// Mitsubishi GX Works2 project: PLC_GROUP2   PLC: FX3G

// global labels: Global1
VAR_GLOBAL
  start_day AT X007 : BOOL;
  Input_Oats AT D1100 : REAL;
  Oats AT D1101 : REAL;
  Input_Pro AT D2100 : REAL;
  Pro AT D2101 : REAL;
  Input_Honey AT D3100 : REAL;
  Honey AT D3101 : REAL;
  work_on AT Y000 : BOOL;
  work_off AT M0 : BOOL;
  end_pack AT M10 : BOOL;
END_VAR
VAR_GLOBAL CONSTANT
  classic_min_pro : REAL := 160;
  classic_min_honey : REAL := 120;
END_VAR
VAR_GLOBAL
  start_mix AT X003 : BOOL;
  Classic AT M16 : BOOL;
  Protein AT M18 : BOOL;
  cannot_mix AT M1 : BOOL;
END_VAR
VAR_GLOBAL CONSTANT
  normalizer : INT := 400;
  max_classic : REAL := 5;
END_VAR
VAR_GLOBAL
  timer_mix_5 AT TC1 : BOOL;
  timer_mix_finish AT TS1 : BOOL;
  mixing AT Y003 : BOOL;
END_VAR
VAR_GLOBAL CONSTANT
  sub_400 : REAL := 400.0;
  sub_160 : REAL := 160.0;
  sub_120 : REAL := 120.0;
  sub_240 : REAL := 240.0;
  sub_320 : REAL := 320.0;
END_VAR
VAR_GLOBAL
  mix_finish AT M8 : BOOL;
  start_bake AT X002 : BOOL;
  finish_bake AT M12 : BOOL;
  timer_bake_classic AT TC2 : BOOL;
END_VAR
VAR_GLOBAL CONSTANT
  four_sec : INT := 40;
END_VAR
VAR_GLOBAL
  timer_bake_pro AT TC3 : BOOL;
END_VAR
VAR_GLOBAL CONSTANT
  five_sec : INT := 50;
END_VAR
VAR_GLOBAL
  timer_bake_classic_finish AT TS2 : BOOL;
  timer_bake_pro_finish AT TS3 : BOOL;
  bake_in_process AT M20 : BOOL;
  timer_bake1 AT TC4 : BOOL;
END_VAR
VAR_GLOBAL CONSTANT
  flashing : INT := 005;
END_VAR
VAR_GLOBAL
  timer_bake1_finish AT TS4 : BOOL;
  lamp1 AT Y001 : BOOL;
  timer_bake2 AT TC5 : BOOL;
  lamp2 AT Y002 : BOOL;
  timer_bake2_finish AT TS5 : BOOL;
  start_pack AT X006 : BOOL;
  pack_hatif AT X000 : BOOL;
  counter_pack AT CC1 : BOOL;
END_VAR
VAR_GLOBAL CONSTANT
  eight_hatifim : INT := 8;
END_VAR
VAR_GLOBAL
  hatifim_packed AT CN1 : INT;
END_VAR
VAR_GLOBAL CONSTANT
  zero : INT;
END_VAR
VAR_GLOBAL
  new_pack AT M30 : BOOL;
  lamp4 AT Y004 : BOOL;
  counter_pack_finish AT CS1 : BOOL;
END_VAR
VAR_GLOBAL CONSTANT
  add_one_pack : INT := 1;
END_VAR
VAR_GLOBAL
  emergency AT X005 : BOOL;
END_VAR
VAR_GLOBAL CONSTANT
  const_40 : REAL := 40;
END_VAR
VAR_GLOBAL
  storage_output AT D5000 : REAL;
END_VAR
VAR_GLOBAL CONSTANT
  classic_min_oats : REAL := 400;
  min_to_start_oat : REAL := 400;
  min_to_start_pro : REAL := 160;
  min_to_start_honey : REAL := 120;
  protein_min_oats : REAL := 240;
  protein_min_pro : REAL := 320;
  protein_min_honey : REAL := 160;
END_VAR
VAR_GLOBAL
  material_empty AT M2 : BOOL;
END_VAR
VAR_GLOBAL CONSTANT
  divider_ten : INT := 10;
  min_protein : REAL := 6;
END_VAR
VAR_GLOBAL
  analog_output AT D8282 : INT;
  analog_input AT D8280 : INT;
END_VAR
VAR_GLOBAL CONSTANT
  mul_400 : INT := 400;
END_VAR
VAR_GLOBAL
  storage AT D7500 : INT;
  hatif AT D7310 : REAL;
END_VAR

// task Task_01 (event TRUE, interval 0, priority 31): POU_01

PROGRAM POU_01
(* structured ladder/FBD written out as ST: instructions are called as NAME(EN, inputs, outputs); _pN, _eN, _tN stand for wires *)
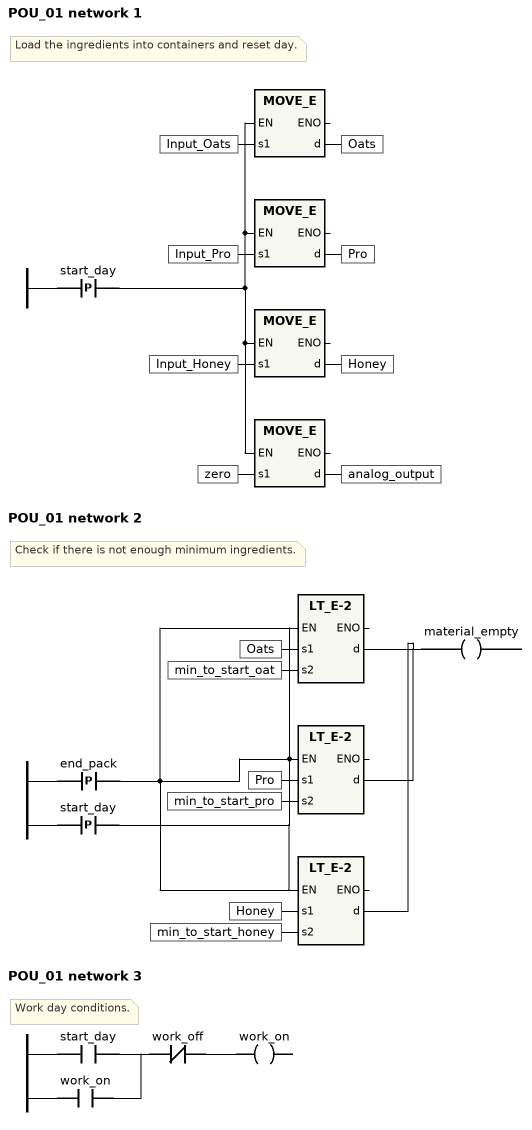
(* network 1 *)
(* Load the ingredients into containers and reset day. *)
_p1 := LDP(TRUE, start_day);
MOVE_E(_p1, Input_Oats, Oats);
MOVE_E(_p1, Input_Pro, Pro);
MOVE_E(_p1, Input_Honey, Honey);
MOVE_E(_p1, zero, analog_output);
(* network 2 *)
(* Check if there is not enough minimum ingredients. *)
_p1 := LDP(TRUE, end_pack) OR LDP(TRUE, start_day);
LT_E(_p1, Oats, min_to_start_oat, _t2);
LT_E(_p1, Pro, min_to_start_pro, _t3);
LT_E(_p1, Honey, min_to_start_honey, _t4);
material_empty := _t2 OR _t3 OR _t4;
(* network 3 *)
(* Work day conditions. *)
work_on := (start_day OR work_on) AND NOT work_off;
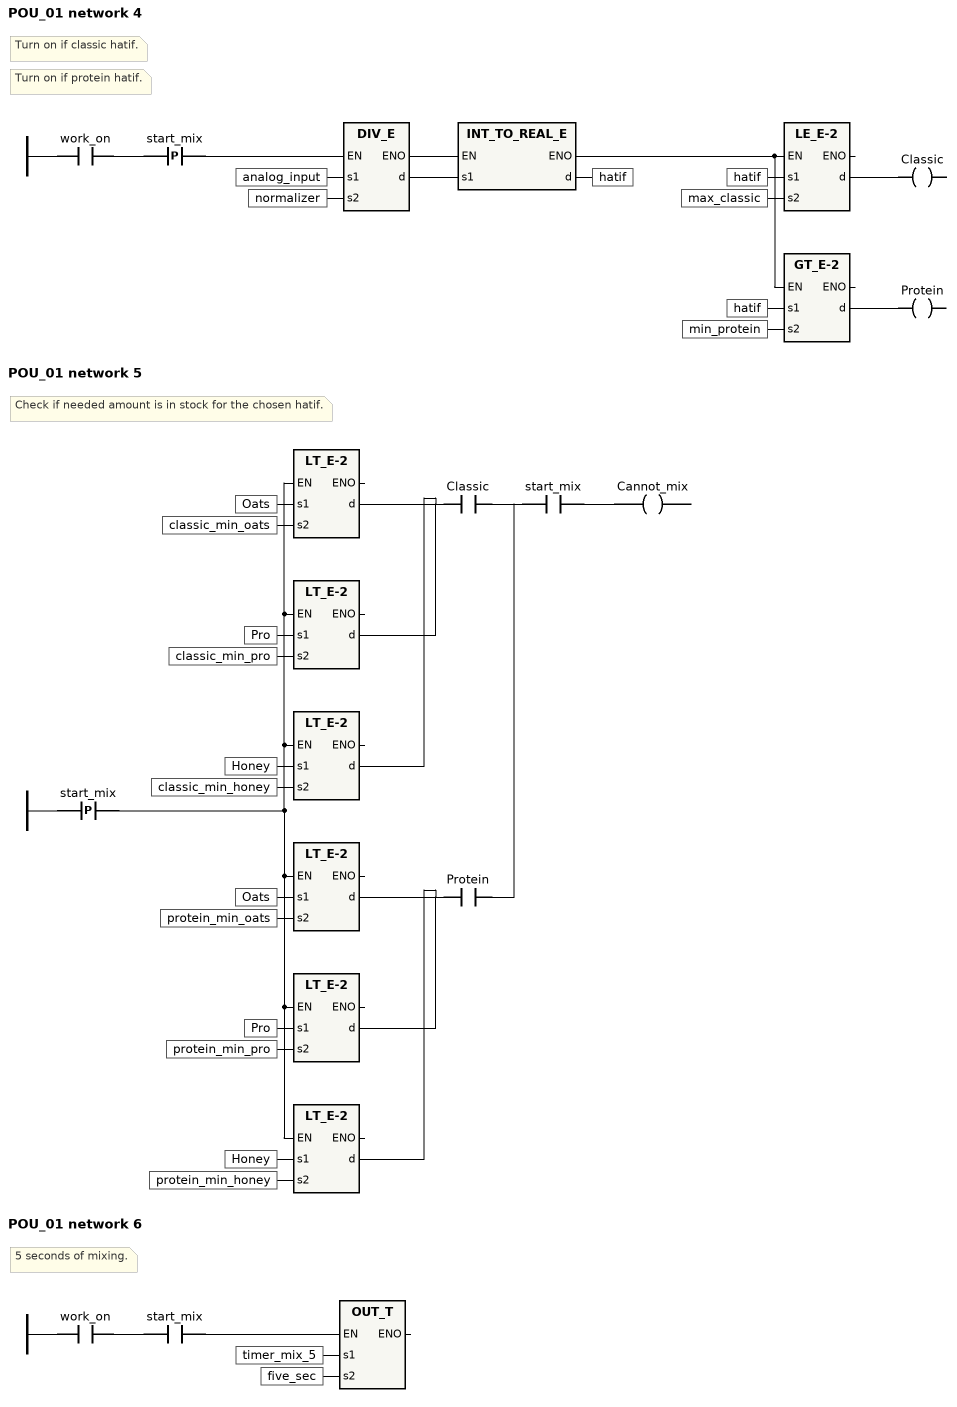
(* network 4 *)
(* Turn on if classic hatif. *)
(* Turn on if protein hatif. *)
_e2 := DIV_E(work_on AND LDP(TRUE, start_mix), analog_input, normalizer, _t1);
_e3 := INT_TO_REAL_E(_e2, _t1, hatif);
LE_E(_e3, hatif, max_classic, _t4);
Classic := _t4;
GT_E(_e3, hatif, min_protein, _t5);
Protein := _t5;
(* network 5 *)
(* Check if needed amount is in stock for the chosen hatif. *)
_p1 := LDP(TRUE, start_mix);
LT_E(_p1, Oats, classic_min_oats, _t2);
LT_E(_p1, Pro, classic_min_pro, _t3);
LT_E(_p1, Honey, classic_min_honey, _t4);
LT_E(_p1, Oats, protein_min_oats, _t5);
LT_E(_p1, Pro, protein_min_pro, _t6);
LT_E(_p1, Honey, protein_min_honey, _t7);
Cannot_mix := (((_t2 OR _t3 OR _t4) AND Classic) OR ((_t5 OR _t6 OR _t7) AND Protein)) AND start_mix;
(* network 6 *)
(* 5 seconds of mixing. *)
OUT_T(work_on AND start_mix, timer_mix_5, five_sec);
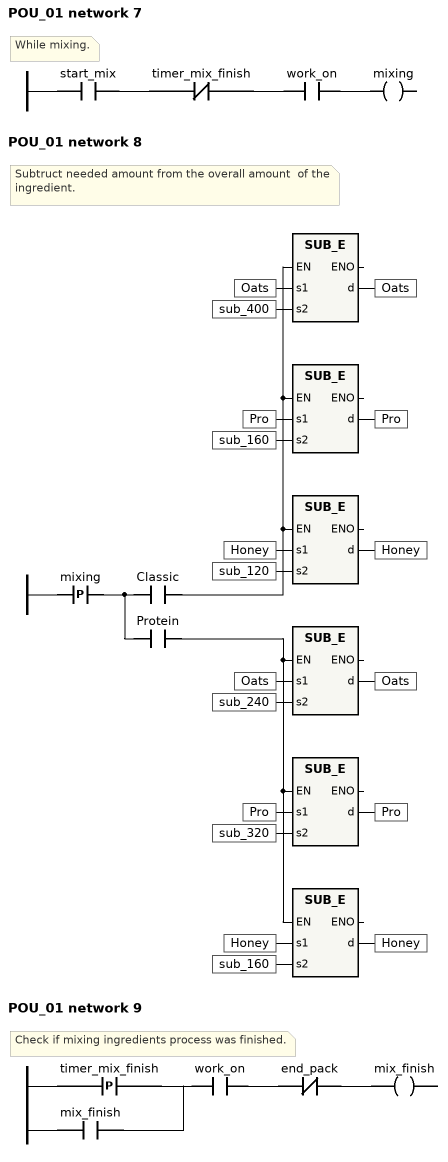
(* network 7 *)
(* While mixing. *)
mixing := start_mix AND NOT timer_mix_finish AND work_on;
(* network 8 *)
(* Subtruct needed amount from the overall amount  of the ingredient. *)
_p1 := LDP(TRUE, mixing);
_p2 := _p1 AND Classic;
SUB_E(_p2, Oats, sub_400, Oats);
SUB_E(_p2, Pro, sub_160, Pro);
SUB_E(_p2, Honey, sub_120, Honey);
_p3 := _p1 AND Protein;
SUB_E(_p3, Oats, sub_240, Oats);
SUB_E(_p3, Pro, sub_320, Pro);
SUB_E(_p3, Honey, sub_160, Honey);
(* network 9 *)
(* Check if mixing ingredients process was finished. *)
mix_finish := ((LDP(TRUE, timer_mix_finish) OR mix_finish) AND work_on) AND NOT end_pack;
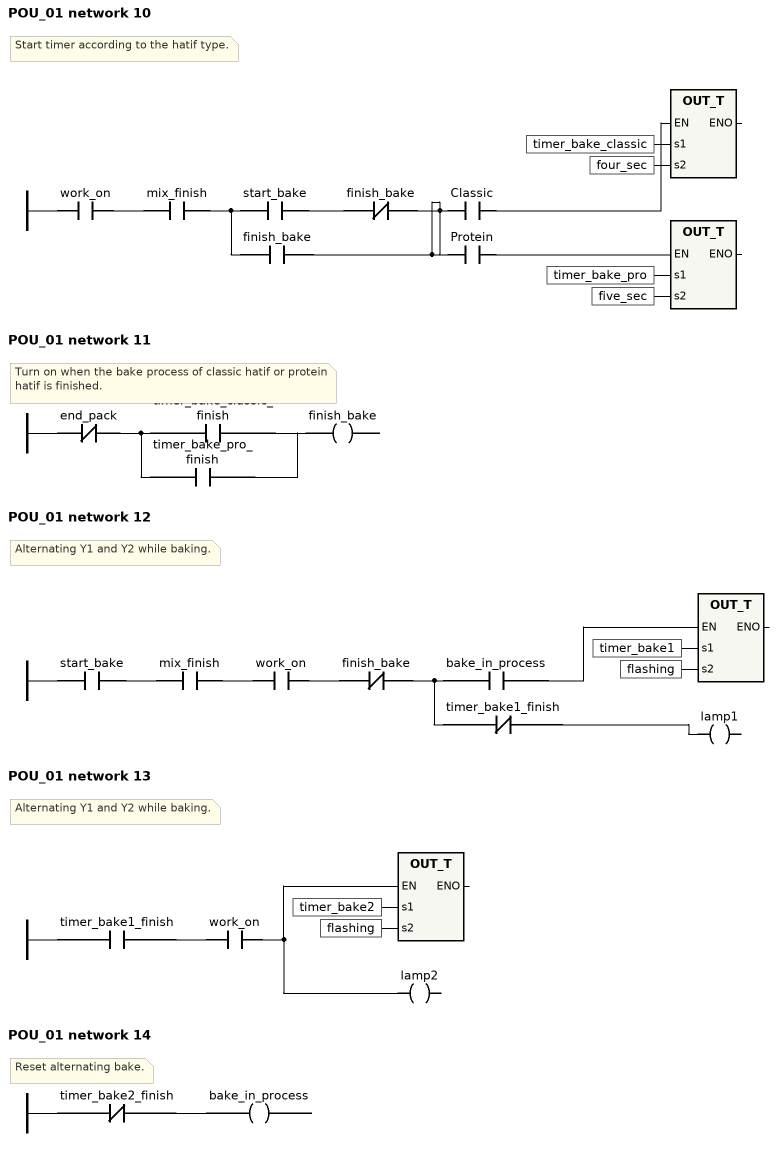
(* network 10 *)
(* Start timer according to the hatif type. *)
_p1 := work_on AND mix_finish;
_p2 := (_p1 AND start_bake AND NOT finish_bake) OR (_p1 AND finish_bake);
OUT_T(_p2 AND Classic, timer_bake_classic, four_sec);
OUT_T(_p2 AND Protein, timer_bake_pro, five_sec);
(* network 11 *)
(* Turn on when the bake process of classic hatif or protein hatif is finished. *)
_p1 := NOT end_pack;
finish_bake := (_p1 AND timer_bake_classic_finish) OR (_p1 AND timer_bake_pro_finish);
(* network 12 *)
(* Alternating Y1 and Y2 while baking. *)
_p1 := start_bake AND mix_finish AND work_on AND NOT finish_bake;
OUT_T(_p1 AND bake_in_process, timer_bake1, flashing);
lamp1 := _p1 AND NOT timer_bake1_finish;
(* network 13 *)
(* Alternating Y1 and Y2 while baking. *)
_p1 := timer_bake1_finish AND work_on;
OUT_T(_p1, timer_bake2, flashing);
lamp2 := _p1;
(* network 14 *)
(* Reset alternating bake. *)
bake_in_process := NOT timer_bake2_finish;
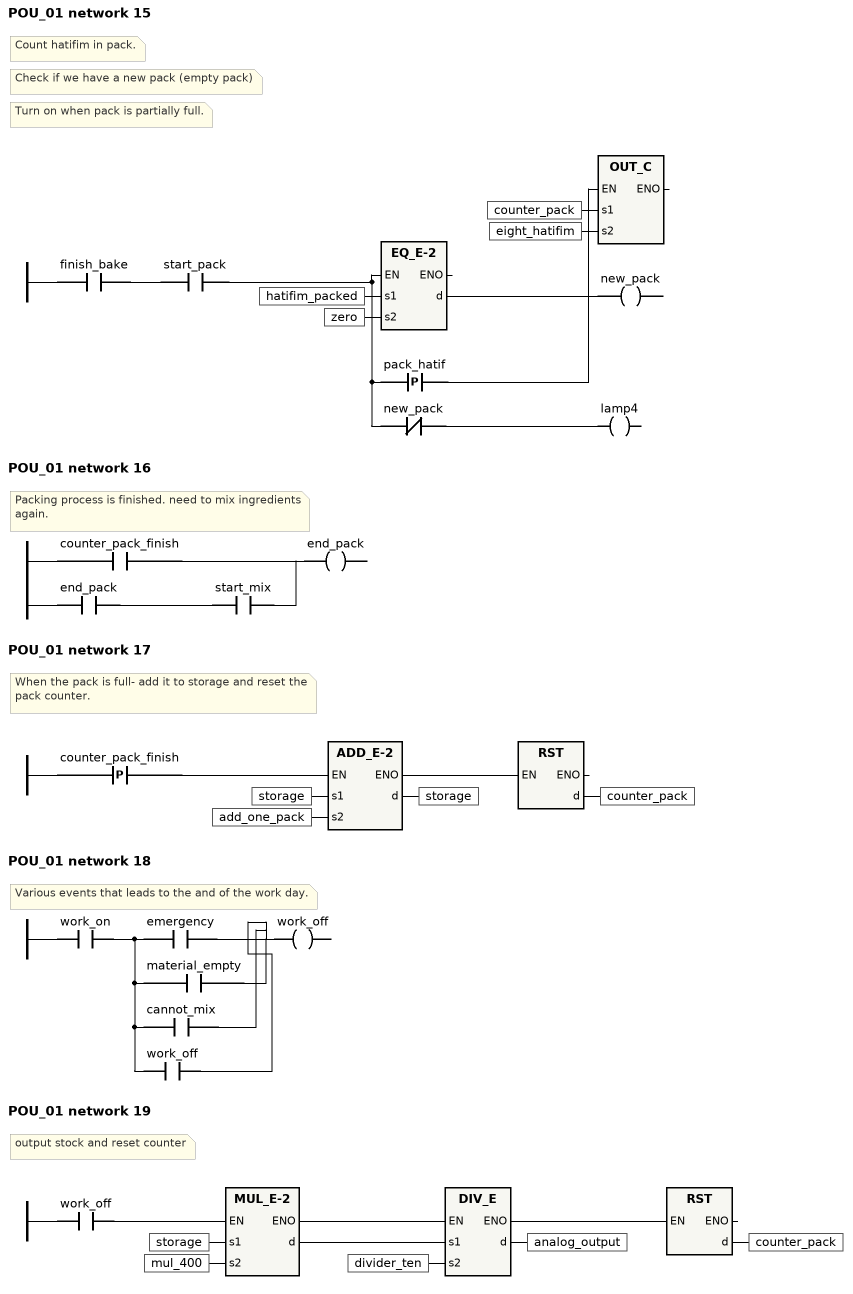
(* network 15 *)
(* Count hatifim in pack. *)
(* Check if we have a new pack (empty pack) *)
(* Turn on when pack is partially full. *)
_p1 := finish_bake AND start_pack;
OUT_C(_p1 AND LDP(TRUE, pack_hatif), counter_pack, eight_hatifim);
EQ_E(_p1, hatifim_packed, zero, _t2);
new_pack := _t2;
lamp4 := _p1 AND NOT new_pack;
(* network 16 *)
(* Packing process is finished. need to mix ingredients again. *)
end_pack := counter_pack_finish OR (end_pack AND start_mix);
(* network 17 *)
(* When the pack is full- add it to storage and reset the pack counter. *)
_e1 := ADD_E(LDP(TRUE, counter_pack_finish), storage, add_one_pack, storage);
RST(_e1, counter_pack);
(* network 18 *)
(* Various events that leads to the and of the work day. *)
work_off := (work_on AND emergency) OR (work_on AND material_empty) OR (work_on AND cannot_mix) OR (work_on AND work_off);
(* network 19 *)
(* output stock and reset counter *)
_e2 := MUL_E(work_off, storage, mul_400, _t1);
_e3 := DIV_E(_e2, _t1, divider_ten, analog_output);
RST(_e3, counter_pack);
END_PROGRAM
